// TwinCAT 3 PLC project OEF_4
// ProgramVersion: 3.1.4024.0
// libraries:
//   Tc2_Standard, * (Beckhoff Automation GmbH)
//   Tc2_System, * (Beckhoff Automation GmbH)
//   Tc3_Module, * (Beckhoff Automation GmbH)
// project tree:
//   / PlcTask.TcTTO
//   POUs/ MAIN.TcPOU
// (motion and I/O tree: see PLC project oef_1)
// real-time tasks:
//   TASK PlcTask: cycle T#10ms, priority 20, ADS port 350
//   TASK PlcTask1: cycle T#10ms, priority 21, ADS port 351
//   TASK PlcTask2: cycle T#10ms, priority 22, ADS port 352
//   TASK PlcTask3: cycle T#10ms, priority 23, ADS port 353
//   TASK PlcTask4: cycle T#10ms, priority 24, ADS port 354
//   TASK PlcTask5: cycle T#10ms, priority 25, ADS port 355
//   TASK PlcTask6: cycle T#10ms, priority 26, ADS port 356
// variable links:
//   OEF_4/OEF_4 Instance <-> Device 1 (EtherCAT)/Term 1 (EK1200)/Term 2 (EL1008)
//     PlcTask Inputs/MAIN.bKnop <-> Channel 1/Input
//   OEF_4/OEF_4 Instance <-> Device 1 (EtherCAT)/Term 1 (EK1200)/Term 3 (EL2008)
//     PlcTask Outputs/MAIN.bLED1 <-> Channel 1/Output

CONFIGURATION OEF_4
    RESOURCE PLC ON TwinCAT3
        TASK PlcTask(INTERVAL := T#10ms, PRIORITY := 24);
        PROGRAM MAIN WITH PlcTask : MAIN;
    END_RESOURCE
END_CONFIGURATION

// ---- POUs/MAIN.TcPOU
PROGRAM MAIN
VAR
	fbTimer: TOF := (PT := TIME#30S0MS);
	bKnop AT %I*: BOOL := false;
	bLED1 AT %Q*: BOOL := FALSE;
	bBuffer AT %Q*: BOOL := false;
	bToggle AT %Q* : BOOL := FALSE;
	fbTrigger: R_TRIG;
END_VAR

fbTrigger(CLK:= bKnop);
IF fbTimer.Q AND fbTrigger.Q THEN
	fbTimer.PT := T#0S;
ELSIF NOT(fbTimer.Q) AND fbTrigger.Q THEN
	fbTimer.PT := T#3S;	
END_IF
fbTimer(IN:= fbTrigger.Q, Q=> bLED1);

END_PROGRAM
